// TwinCAT 3 PLC project Untitled1
// ProgramVersion: 3.1.4026.16
// CompilerDefines: VISU_USEPROPERTYINFO
// libraries:
//   Tc2_Standard, * (Beckhoff Automation GmbH)
//   Tc2_System, * (Beckhoff Automation GmbH)
//   VisuSymbols, 4.5.0.0 (System)
// project tree:
//   / GlobalTextList.TcGTLO, PlcTask.TcTTO, Visualization Manager.TcVMO (not stored)
//   POUs/ MAIN.TcPOU
//   VISUs/ Visualization.TcVIS

CONFIGURATION Untitled1
    RESOURCE PLC ON TwinCAT3
        TASK PlcTask(INTERVAL := T#10ms, PRIORITY := 20);
        PROGRAM MAIN WITH PlcTask : MAIN;
    END_RESOURCE
END_CONFIGURATION

// ---- POUs/MAIN.TcPOU
PROGRAM MAIN
VAR
	iRBig : REAL := 150;
	iRSmall : REAL := 50;
	rAngle: REAL;
	rAngularVelocity : REAL := 90;
	rSmallX: REAL;
	rSmallY: REAL;
	PI: REAL := 3.14159;
END_VAR

IF iRSmall > (iRBig / 2) THEN
	iRSmall := iRBig/2;
END_IF

rAngle := rAngle + (0.01 * rAngularVelocity);

rSmallX := iRBig + (iRBig - iRSmall)*COS(rAngle * (PI / 180)) - iRSmall;
rSmallY := iRBig + (iRBig - iRSmall)*SIN(rAngle * (PI / 180)) - iRSmall;

END_PROGRAM

// ---- VISUs/Visualization.TcVIS
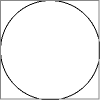
VISUALIZATION Visualization  // 100x100
    Ellipse (0,0 100x100)
        p3560616238: MAIN.iRBig - 50
        p1097714728: ((MAIN.iRBig) / 50 ) * 1000
        p2738717112: MAIN.iRBig - 50
    Ellipse (0,0 100x100)
        p3560616238: MAIN.iRSmall - 50 + MAIN.rSmallX
        p1097714728: ((MAIN.iRSmall) / 50 ) * 1000
        p2738717112: MAIN.iRSmall - 50 + MAIN.rSmallY
END_VISUALIZATION
